TYPE ST_Ifm_RX :
STRUCT
		OutputByte : ARRAY[0..3] OF USINT;
END_STRUCT
END_TYPE

(* stored: Version 1.1.0.1, ProductVersion 3.1.4024.12
   DUT ST_Ifm_RX: Id {c4f2d9a9-7966-420d-8074-cdaccf2ddf04} *)
